Universal Robots PolyScope program: proiecFinalHILT_cri.urp

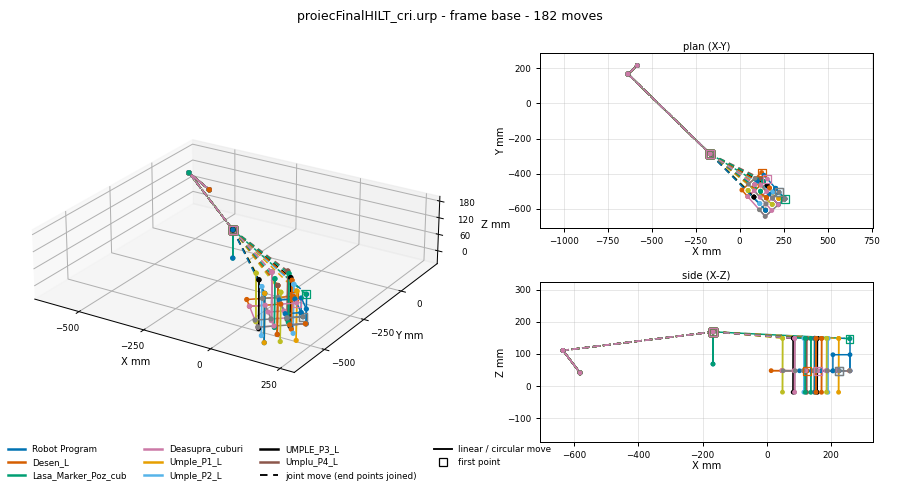
[picture p0: tool path of proiecFinalHILT_cri.urp in frame base, 182 of 182 moves have a stored position in this frame; points joined in program order, loops and branches not executed]
Program proiecFinalHILT_cri (installation=default directory=/home/ur/ursim-current/programs/Setup createdIn=3.15.5.106321 lastSavedIn=3.15.5.106321 robotSerialNumber=2018359999)
Calibrated DH parameters: a=[0, -0.425, -0.39225, 0, 0, 0]; d=[0.089159, 0, 0, 0.10915, 0.09465, 0.0823]; alpha=[1.570796, 0, 0, 1.570796, -1.570796, 0]; deltaTheta=[0, 0, 0, 0, 0, 0]
Robot Program (runOnlyOnce=false)
  MoveL speed 250 mm/s, acceleration 1200 mm/s^2 (useActiveTCP=true) feature=Base
    Waypoint Intermediar_cub: TCP in base x=-167.567 y=-286.499 z=168.811 mm, rx=1.2909 ry=2.8479 rz=-0.0144 rad; joints [39.36, -114.131, 107.649, -83.617, -89.01, -1.87] deg; flange x=-170.167 y=-282.588 z=439.18 mm, rx=1.2909 ry=2.8479 rz=-0.0144 rad
    Waypoint preluare_marker: TCP in base x=-167.81 y=-286.838 z=68.812 mm, rx=1.2909 ry=2.8479 rz=-0.0144 rad; joints [39.38, -113.83, 122.13, -98.4, -89.01, -1.85] deg; flange x=-170.409 y=-282.927 z=339.181 mm, rx=1.2909 ry=2.8479 rz=-0.0144 rad
    Wait Sleep waitTime=0.5
    'G 10'
    Wait Sleep waitTime=0.5
  MoveL speed 250 mm/s, acceleration 1200 mm/s^2 (useActiveTCP=true) feature=Base
    Waypoint ridicare_marker: TCP in base x=-167.568 y=-286.499 z=168.811 mm, rx=1.2909 ry=2.8479 rz=-0.0144 rad; joints [39.36, -114.131, 107.649, -83.617, -89.01, -1.87] deg; flange x=-170.167 y=-282.588 z=439.18 mm, rx=1.2909 ry=2.8479 rz=-0.0144 rad
  MoveJ speed 60 deg/s, acceleration 80 deg/s^2 (useActiveTCP=true)
    Waypoint deasupra_colt_f: TCP in base x=258.142 y=-542.024 z=147.75 mm, rx=1.296 ry=2.8485 rz=0.0145 rad; joints [104.471, -76.071, 76.258, -90.209, -89.13, 63.401] deg; flange x=254.141 y=-542.951 z=418.128 mm, rx=1.296 ry=2.8485 rz=0.0145 rad
  MoveL speed 250 mm/s, acceleration 1200 mm/s^2 (useActiveTCP=true) feature=Base
    Waypoint marker_pe_colt: TCP in base x=257.9 y=-542.363 z=47.75 mm, rx=1.296 ry=2.8485 rz=0.0145 rad; joints [104.44, -74.31, 88.769, -104.48, -89.13, 63.37] deg; flange x=253.899 y=-543.29 z=318.129 mm, rx=1.296 ry=2.8485 rz=0.0145 rad
  If digital_in[1] == True
    Call Desen_L
    Call Lasa_Marker_Poz_cub
    Call Deasupra_cuburi
    Call Umple_P1_L
    Call Umple_P2_L
    Call UMPLE_P3_L
    Call Umplu_P4_L
    Call Umplu_P5_L
    Call Umplu_P6_L
  If digital_in[2] ==  True
    Call Desen_i
    Call Lasa_Marker_Poz_cub
    Call Deasupra_cuburi
    Call Umple_P1_L
    Call Umplu_p2_i
    Call Umplu_p3_i
  If digital_in[3] ==  True
    Call Desen_H
    Call Lasa_Marker_Poz_cub
    Call Deasupra_cuburi
    Call Umple_P1_L
    Call Umple_P2_L
    Call UMPLE_P3_L
    Call Umple_P4_H
    Call Umple_P5_H
    Call Umple_P6_H
    Call Umple_P7_H
  If digital_in[5] ==  True
    Call Desen_T
    Call Lasa_Marker_Poz_cub
    Call Deasupra_cuburi
    Call Umple_P1_L
    Call Umple_P2_T
    Call Umple_p3_T
    Call Umplu_p4_t
    Call Umplu_p5_T
    Call Umple_P6_T
SubProgram -> Umple_P7_H
SubProgram -> Umple_P6_H
SubProgram -> Umple_P5_H
SubProgram -> Umple_P4_H
SubProgram -> Umple_P6_T
SubProgram -> Umplu_p5_T
SubProgram -> Umplu_p4_t
SubProgram -> Umple_p3_T
SubProgram -> Umple_P2_T
SubProgram -> Desen_H
SubProgram -> Desen_T
SubProgram -> Umplu_p3_i
SubProgram -> Umplu_p2_i
SubProgram -> Desen_i
SubProgram -> Umplu_P6_L
SubProgram -> Umplu_P5_L
SubProgram -> Umplu_P4_L
SubProgram -> UMPLE_P3_L
SubProgram -> Umple_P2_L
SubProgram -> Umple_P1_L
SubProgram -> Deasupra_cuburi
SubProgram -> Lasa_Marker_Poz_cub
SubProgram -> Desen_L
SubProgram Desen_L (keepSynchronizedWithDisk=false)
  MoveL speed 250 mm/s, acceleration 1200 mm/s^2 (useActiveTCP=true) feature=Base
    Waypoint exterior_L: TCP in base x=125.172 y=-392.753 z=47.565 mm, rx=1.296 ry=2.8485 rz=0.0145 rad; joints [91.565, -100.156, 115.983, -105.654, -89.147, 50.493] deg; flange x=121.171 y=-393.68 z=317.944 mm, rx=1.296 ry=2.8485 rz=0.0145 rad
  MoveL speed 250 mm/s, acceleration 1200 mm/s^2 (useActiveTCP=true) feature=Base
    Waypoint Exterior_L2: TCP in base x=12.964 y=-492.297 z=48.174 mm, rx=1.296 ry=2.8485 rz=0.0145 rad; joints [78.123, -88.524, 105.201, -106.311, -89.211, 37.05] deg; flange x=8.963 y=-493.224 z=318.552 mm, rx=1.296 ry=2.8485 rz=0.0145 rad
  MoveL speed 250 mm/s, acceleration 1200 mm/s^2 (useActiveTCP=true) feature=Base
    Waypoint Exterior_L3: TCP in base x=46.146 y=-529.7 z=48.22 mm, rx=1.296 ry=2.8485 rz=0.0145 rad; joints [82.58, -83.248, 99.507, -105.954, -89.185, 41.507] deg; flange x=42.145 y=-530.627 z=318.599 mm, rx=1.296 ry=2.8485 rz=0.0145 rad
  MoveL speed 250 mm/s, acceleration 1200 mm/s^2 (useActiveTCP=true) feature=Base
    Waypoint Interior_L: TCP in base x=120.04 y=-464.145 z=47.819 mm, rx=1.296 ry=2.8485 rz=0.0145 rad; joints [90.697, -90.465, 107.261, -106.61, -89.15, 49.626] deg; flange x=116.039 y=-465.073 z=318.198 mm, rx=1.296 ry=2.8485 rz=0.0145 rad
  MoveL speed 250 mm/s, acceleration 1200 mm/s^2 (useActiveTCP=true) feature=Base
    Waypoint Interior_L2: TCP in base x=219.586 y=-576.353 z=47.958 mm, rx=1.296 ry=2.8485 rz=0.0145 rad; joints [100.158, -72.107, 85.808, -103.657, -89.131, 59.087] deg; flange x=215.585 y=-577.28 z=318.337 mm, rx=1.296 ry=2.8485 rz=0.0145 rad
  MoveL speed 250 mm/s, acceleration 1200 mm/s^2 (useActiveTCP=true) feature=Base
    Waypoint Interior_L3: TCP in base x=256.233 y=-543.842 z=47.759 mm, rx=1.296 ry=2.8485 rz=0.0145 rad; joints [104.247, -74.225, 88.656, -104.449, -89.13, 63.177] deg; flange x=252.231 y=-544.769 z=318.138 mm, rx=1.296 ry=2.8485 rz=0.0145 rad
SubProgram Lasa_Marker_Poz_cub (keepSynchronizedWithDisk=false)
  MoveL speed 250 mm/s, acceleration 1200 mm/s^2 (useActiveTCP=true) feature=Base
    Waypoint DeasupraFoaie: TCP in base x=256.475 y=-543.503 z=147.759 mm, rx=1.296 ry=2.8485 rz=0.0145 rad; joints [104.278, -75.981, 76.142, -90.18, -89.13, 63.208] deg; flange x=252.473 y=-544.43 z=418.137 mm, rx=1.296 ry=2.8485 rz=0.0145 rad
  MoveJ speed 60 deg/s, acceleration 80 deg/s^2 (useActiveTCP=true)
    Waypoint DeasupraMarker: TCP in base x=-167.557 y=-286.49 z=168.795 mm, rx=1.2909 ry=2.8479 rz=-0.0143 rad; joints [39.36, -114.132, 107.651, -83.617, -89.01, -1.87] deg; flange x=-170.163 y=-282.585 z=439.164 mm, rx=1.2909 ry=2.8479 rz=-0.0143 rad
  MoveL speed 250 mm/s, acceleration 1200 mm/s^2 (useActiveTCP=true) feature=Base
    Waypoint LasaMarker: TCP in base x=-167.799 y=-286.829 z=68.796 mm, rx=1.2909 ry=2.8479 rz=-0.0143 rad; joints [39.38, -113.83, 122.132, -98.4, -89.01, -1.85] deg; flange x=-170.405 y=-282.924 z=339.165 mm, rx=1.2909 ry=2.8479 rz=-0.0143 rad
    Wait Sleep waitTime=0.5
    'G 40'
    Wait Sleep waitTime=0.5
  MoveL speed 250 mm/s, acceleration 1200 mm/s^2 (useActiveTCP=true) feature=Base
    Waypoint DeasupraMarker2: TCP in base x=-167.557 y=-286.49 z=168.795 mm, rx=1.2909 ry=2.8479 rz=-0.0143 rad; joints [39.36, -114.132, 107.651, -83.617, -89.01, -1.87] deg; flange x=-170.163 y=-282.585 z=439.164 mm, rx=1.2909 ry=2.8479 rz=-0.0143 rad
    Wait Sleep waitTime=0.5
    'G80'
SubProgram Deasupra_cuburi (keepSynchronizedWithDisk=false)
  MoveL speed 250 mm/s, acceleration 1200 mm/s^2 (useActiveTCP=true) feature=Base
    Waypoint DeasupraMarker2: TCP in base x=-167.557 y=-286.49 z=168.795 mm, rx=1.2909 ry=2.8479 rz=-0.0143 rad; joints [39.36, -114.132, 107.651, -83.617, -89.01, -1.87] deg; flange x=-170.163 y=-282.585 z=439.164 mm, rx=1.2909 ry=2.8479 rz=-0.0143 rad
  MoveJ speed 60 deg/s, acceleration 80 deg/s^2 (useActiveTCP=true)
    Waypoint poz_intermcub: TCP in base x=-634.049 y=166.753 z=111.017 mm, rx=1.0761 ry=2.3886 rz=1.0065 rad; joints [-7.715, -31.545, 17.047, -40.87, -122.454, -38.841] deg; flange x=-782.032 y=40.366 z=298.765 mm, rx=1.0761 ry=2.3886 rz=1.0065 rad
  MoveL speed 250 mm/s, acceleration 1200 mm/s^2 (useActiveTCP=true) feature=Base
    Waypoint prindere_cub: TCP in base x=-580.967 y=215.041 z=41.371 mm, rx=1.0761 ry=2.3886 rz=1.0065 rad; joints [-11.8, -45.21, 53.1, -65.52, -124.71, -42.93] deg; flange x=-728.95 y=88.654 z=229.118 mm, rx=1.0761 ry=2.3886 rz=1.0065 rad
    Wait Sleep waitTime=0.5
    'G40'
  MoveL speed 250 mm/s, acceleration 1200 mm/s^2 (useActiveTCP=true) feature=Base
    Waypoint poz_intermcub: TCP in base x=-634.049 y=166.753 z=111.017 mm, rx=1.0761 ry=2.3886 rz=1.0065 rad; joints [-7.715, -31.545, 17.047, -40.87, -122.454, -38.841] deg; flange x=-782.032 y=40.366 z=298.765 mm, rx=1.0761 ry=2.3886 rz=1.0065 rad
    Wait Sleep waitTime=0.5
SubProgram Umple_P1_L (keepSynchronizedWithDisk=false)
  MoveJ speed 60 deg/s, acceleration 80 deg/s^2 (useActiveTCP=true)
    Waypoint Intermediar_cub: TCP in base x=-167.567 y=-286.499 z=168.811 mm, rx=1.2909 ry=2.8479 rz=-0.0144 rad; joints [39.36, -114.131, 107.649, -83.617, -89.01, -1.87] deg; flange x=-170.167 y=-282.588 z=439.18 mm, rx=1.2909 ry=2.8479 rz=-0.0144 rad
    Wait Sleep waitTime=0.5
  MoveJ speed 60 deg/s, acceleration 80 deg/s^2 (useActiveTCP=true)
    Waypoint cb_deas_fo_cent: TCP in base x=222.984 y=-540.437 z=148.398 mm, rx=2.9837 ry=0.9733 rz=-0.0052 rad; joints [101.765, -78.264, 78.922, -90.858, -90.17, 155.632] deg; flange x=223.577 y=-539.348 z=418.805 mm, rx=2.9837 ry=0.9733 rz=-0.0052 rad
    Wait Sleep waitTime=0.5
  MoveL speed 250 mm/s, acceleration 1200 mm/s^2 (useActiveTCP=true) feature=Base
    Waypoint las_1_cub_foaie: TCP in base x=222.579 y=-541.004 z=-18.947 mm, rx=2.9837 ry=0.9733 rz=-0.0052 rad; joints [101.714, -73.294, 97.815, -114.721, -90.17, 155.581] deg; flange x=223.172 y=-539.915 z=251.46 mm, rx=2.9837 ry=0.9733 rz=-0.0052 rad
    Wait Sleep waitTime=0.5
    'G 80'
  MoveL speed 250 mm/s, acceleration 1200 mm/s^2 (useActiveTCP=true) feature=Base
    Waypoint Deasupra_foaiee: TCP in base x=222.984 y=-540.437 z=148.398 mm, rx=2.9837 ry=0.9733 rz=-0.0052 rad; joints [101.765, -78.264, 78.922, -90.858, -90.17, 155.632] deg; flange x=223.577 y=-539.348 z=418.805 mm, rx=2.9837 ry=0.9733 rz=-0.0052 rad
SubProgram Umple_P2_L (keepSynchronizedWithDisk=false)
  MoveJ speed 60 deg/s, acceleration 80 deg/s^2 (useActiveTCP=true)
    Waypoint interm_P2: TCP in base x=-167.567 y=-286.499 z=168.811 mm, rx=1.2909 ry=2.8479 rz=-0.0144 rad; joints [39.36, -114.131, 107.649, -83.617, -89.01, -1.87] deg; flange x=-170.167 y=-282.588 z=439.18 mm, rx=1.2909 ry=2.8479 rz=-0.0144 rad
    Wait Sleep waitTime=0.5
  MoveJ speed 60 deg/s, acceleration 80 deg/s^2 (useActiveTCP=true)
    Waypoint DEAS_cub_C2_L: TCP in base x=-634.049 y=166.753 z=111.017 mm, rx=1.0761 ry=2.3886 rz=1.0065 rad; joints [-7.715, -31.545, 17.047, -40.87, -122.454, -38.841] deg; flange x=-782.032 y=40.366 z=298.765 mm, rx=1.0761 ry=2.3886 rz=1.0065 rad
    Wait Sleep waitTime=0.5
  MoveL speed 250 mm/s, acceleration 1200 mm/s^2 (useActiveTCP=true) feature=Base
    Waypoint prel_c2_L: TCP in base x=-580.967 y=215.041 z=41.371 mm, rx=1.0761 ry=2.3886 rz=1.0065 rad; joints [-11.8, -45.21, 53.1, -65.52, -124.71, -42.93] deg; flange x=-728.95 y=88.654 z=229.118 mm, rx=1.0761 ry=2.3886 rz=1.0065 rad
    Wait Sleep waitTime=0.5
    'G40'
  MoveL speed 250 mm/s, acceleration 1200 mm/s^2 (useActiveTCP=true) feature=Base
    Waypoint deas_c2_L: TCP in base x=-634.049 y=166.753 z=111.017 mm, rx=1.0761 ry=2.3886 rz=1.0065 rad; joints [-7.715, -31.545, 17.047, -40.87, -122.454, -38.841] deg; flange x=-782.032 y=40.366 z=298.765 mm, rx=1.0761 ry=2.3886 rz=1.0065 rad
    Wait Sleep waitTime=0.5
  MoveJ speed 60 deg/s, acceleration 80 deg/s^2 (useActiveTCP=true)
    Waypoint INTERM: TCP in base x=-167.567 y=-286.499 z=168.811 mm, rx=1.2909 ry=2.8479 rz=-0.0144 rad; joints [39.36, -114.131, 107.649, -83.617, -89.01, -1.87] deg; flange x=-170.167 y=-282.588 z=439.18 mm, rx=1.2909 ry=2.8479 rz=-0.0144 rad
    Wait Sleep waitTime=0.5
  MoveJ speed 60 deg/s, acceleration 80 deg/s^2 (useActiveTCP=true)
    Waypoint DEAS_P2_L_FOAIE: TCP in base x=189.802 y=-503.035 z=148.352 mm, rx=2.9837 ry=0.9733 rz=-0.0052 rad; joints [99.066, -84.782, 86.489, -91.915, -90.16, 152.933] deg; flange x=190.395 y=-501.946 z=418.759 mm, rx=2.9837 ry=0.9733 rz=-0.0052 rad
    Wait Sleep waitTime=0.5
  MoveL speed 250 mm/s, acceleration 1200 mm/s^2 (useActiveTCP=true) feature=Base
    Waypoint LAS_P2_L_FOAIE: TCP in base x=189.397 y=-503.602 z=-18.994 mm, rx=2.9837 ry=0.9733 rz=-0.0052 rad; joints [99.013, -79.253, 105.478, -116.434, -90.16, 152.88] deg; flange x=189.99 y=-502.512 z=251.414 mm, rx=2.9837 ry=0.9733 rz=-0.0052 rad
    Wait Sleep waitTime=0.5
    'G 80'
  MoveL speed 250 mm/s, acceleration 1200 mm/s^2 (useActiveTCP=true) feature=Base
    Waypoint DEAS_P2_L: TCP in base x=189.802 y=-503.035 z=148.352 mm, rx=2.9837 ry=0.9733 rz=-0.0052 rad; joints [99.067, -84.782, 86.489, -91.915, -90.16, 152.933] deg; flange x=190.395 y=-501.945 z=418.759 mm, rx=2.9837 ry=0.9733 rz=-0.0052 rad
SubProgram UMPLE_P3_L (keepSynchronizedWithDisk=false)
  MoveJ speed 60 deg/s, acceleration 80 deg/s^2 (useActiveTCP=true)
    Waypoint INTERM_P3: TCP in base x=-167.567 y=-286.499 z=168.811 mm, rx=1.2909 ry=2.8479 rz=-0.0144 rad; joints [39.36, -114.131, 107.649, -83.617, -89.01, -1.87] deg; flange x=-170.167 y=-282.588 z=439.18 mm, rx=1.2909 ry=2.8479 rz=-0.0144 rad
    Wait Sleep waitTime=0.5
  MoveJ speed 60 deg/s, acceleration 80 deg/s^2 (useActiveTCP=true)
    Waypoint DEAS_C3_L: TCP in base x=-634.049 y=166.753 z=111.017 mm, rx=1.0761 ry=2.3886 rz=1.0065 rad; joints [-7.715, -31.545, 17.047, -40.87, -122.454, -38.841] deg; flange x=-782.032 y=40.366 z=298.765 mm, rx=1.0761 ry=2.3886 rz=1.0065 rad
    Wait Sleep waitTime=0.5
  MoveL speed 250 mm/s, acceleration 1200 mm/s^2 (useActiveTCP=true) feature=Base
    Waypoint PREL_C3_L: TCP in base x=-580.967 y=215.041 z=41.371 mm, rx=1.0761 ry=2.3886 rz=1.0065 rad; joints [-11.8, -45.21, 53.1, -65.52, -124.71, -42.93] deg; flange x=-728.95 y=88.654 z=229.118 mm, rx=1.0761 ry=2.3886 rz=1.0065 rad
    Wait Sleep waitTime=0.5
    'G40'
  MoveL speed 250 mm/s, acceleration 1200 mm/s^2 (useActiveTCP=true) feature=Base
    Waypoint DEAS_C3_LL: TCP in base x=-634.049 y=166.753 z=111.017 mm, rx=1.0761 ry=2.3886 rz=1.0065 rad; joints [-7.715, -31.545, 17.047, -40.87, -122.454, -38.841] deg; flange x=-782.032 y=40.366 z=298.765 mm, rx=1.0761 ry=2.3886 rz=1.0065 rad
    Wait Sleep waitTime=0.5
  MoveJ speed 60 deg/s, acceleration 80 deg/s^2 (useActiveTCP=true)
    Waypoint INTERMMM: TCP in base x=-167.567 y=-286.499 z=168.811 mm, rx=1.2909 ry=2.8479 rz=-0.0144 rad; joints [39.36, -114.131, 107.649, -83.617, -89.01, -1.87] deg; flange x=-170.167 y=-282.588 z=439.18 mm, rx=1.2909 ry=2.8479 rz=-0.0144 rad
    Wait Sleep waitTime=0.5
  MoveJ speed 60 deg/s, acceleration 80 deg/s^2 (useActiveTCP=true)
    Waypoint DEAS_P3_L_FOAIE: TCP in base x=156.62 y=-465.632 z=148.305 mm, rx=2.9837 ry=0.9733 rz=-0.0052 rad; joints [95.863, -91.188, 93.147, -92.177, -90.149, 149.73] deg; flange x=157.213 y=-464.543 z=418.713 mm, rx=2.9837 ry=0.9733 rz=-0.0052 rad
    Wait Sleep waitTime=0.5
  MoveL speed 250 mm/s, acceleration 1200 mm/s^2 (useActiveTCP=true) feature=Base
    Waypoint LAS_P3_L_FOAIE: TCP in base x=156.215 y=-466.199 z=-19.04 mm, rx=2.9837 ry=0.9733 rz=-0.0052 rad; joints [95.808, -85.301, 112.521, -117.438, -90.148, 149.675] deg; flange x=156.808 y=-465.11 z=251.367 mm, rx=2.9837 ry=0.9733 rz=-0.0052 rad
    Wait Sleep waitTime=0.5
    'G 80'
  MoveL speed 250 mm/s, acceleration 1200 mm/s^2 (useActiveTCP=true) feature=Base
    Waypoint DEASUPRA_P3_L: TCP in base x=156.62 y=-465.632 z=148.305 mm, rx=2.9837 ry=0.9733 rz=-0.0052 rad; joints [95.863, -91.188, 93.147, -92.177, -90.149, 149.73] deg; flange x=157.213 y=-464.543 z=418.713 mm, rx=2.9837 ry=0.9733 rz=-0.0052 rad
SubProgram Umplu_P4_L (keepSynchronizedWithDisk=false)
  MoveJ speed 60 deg/s, acceleration 80 deg/s^2 (useActiveTCP=true)
    Waypoint INTERM_P4: TCP in base x=-167.567 y=-286.499 z=168.811 mm, rx=1.2909 ry=2.8479 rz=-0.0144 rad; joints [39.36, -114.131, 107.649, -83.617, -89.01, -1.87] deg; flange x=-170.167 y=-282.588 z=439.18 mm, rx=1.2909 ry=2.8479 rz=-0.0144 rad
    Wait Sleep waitTime=0.5
  MoveJ speed 60 deg/s, acceleration 80 deg/s^2 (useActiveTCP=true)
    Waypoint DEAS_C4_L: TCP in base x=-634.049 y=166.753 z=111.017 mm, rx=1.0761 ry=2.3886 rz=1.0065 rad; joints [-7.715, -31.545, 17.047, -40.87, -122.454, -38.841] deg; flange x=-782.032 y=40.366 z=298.765 mm, rx=1.0761 ry=2.3886 rz=1.0065 rad
    Wait Sleep waitTime=0.5
  MoveL speed 250 mm/s, acceleration 1200 mm/s^2 (useActiveTCP=true) feature=Base
    Waypoint PREL_C4_L: TCP in base x=-580.967 y=215.041 z=41.371 mm, rx=1.0761 ry=2.3886 rz=1.0065 rad; joints [-11.8, -45.21, 53.1, -65.52, -124.71, -42.93] deg; flange x=-728.95 y=88.654 z=229.118 mm, rx=1.0761 ry=2.3886 rz=1.0065 rad
    Wait Sleep waitTime=0.5
    'G40'
  MoveL speed 250 mm/s, acceleration 1200 mm/s^2 (useActiveTCP=true) feature=Base
    Waypoint DEAS_C4_LL: TCP in base x=-634.049 y=166.753 z=111.017 mm, rx=1.0761 ry=2.3886 rz=1.0065 rad; joints [-7.715, -31.545, 17.047, -40.87, -122.454, -38.841] deg; flange x=-782.032 y=40.366 z=298.765 mm, rx=1.0761 ry=2.3886 rz=1.0065 rad
    Wait Sleep waitTime=0.5
  MoveJ speed 60 deg/s, acceleration 80 deg/s^2 (useActiveTCP=true)
    Waypoint INTER: TCP in base x=-167.567 y=-286.499 z=168.811 mm, rx=1.2909 ry=2.8479 rz=-0.0144 rad; joints [39.36, -114.131, 107.649, -83.617, -89.01, -1.87] deg; flange x=-170.167 y=-282.588 z=439.18 mm, rx=1.2909 ry=2.8479 rz=-0.0144 rad
    Wait Sleep waitTime=0.5
  MoveJ speed 60 deg/s, acceleration 80 deg/s^2 (useActiveTCP=true)
    Waypoint DEAS_P4_L_FOAIE: TCP in base x=123.438 y=-428.23 z=148.259 mm, rx=2.9837 ry=0.9733 rz=-0.0052 rad; joints [92.012, -97.554, 98.997, -91.67, -90.134, 145.879] deg; flange x=124.031 y=-427.14 z=418.666 mm, rx=2.9837 ry=0.9733 rz=-0.0052 rad
    Wait Sleep waitTime=0.5
  MoveL speed 250 mm/s, acceleration 1200 mm/s^2 (useActiveTCP=true) feature=Base
    Waypoint LAS_P4_L_FOAIE: TCP in base x=123.033 y=-428.796 z=-19.086 mm, rx=2.9837 ry=0.9733 rz=-0.0052 rad; joints [91.956, -91.539, 118.98, -117.667, -90.133, 145.823] deg; flange x=123.626 y=-427.707 z=251.321 mm, rx=2.9837 ry=0.9733 rz=-0.0052 rad
    Wait Sleep waitTime=0.5
    'G 80'
  MoveL speed 250 mm/s, acceleration 1200 mm/s^2 (useActiveTCP=true) feature=Base
    Waypoint DEAS_P4_L: TCP in base x=123.438 y=-428.23 z=148.259 mm, rx=2.9837 ry=0.9733 rz=-0.0052 rad; joints [92.012, -97.554, 98.997, -91.67, -90.134, 145.879] deg; flange x=124.031 y=-427.14 z=418.666 mm, rx=2.9837 ry=0.9733 rz=-0.0052 rad
SubProgram Umplu_P5_L (keepSynchronizedWithDisk=false)
  MoveJ speed 60 deg/s, acceleration 80 deg/s^2 (useActiveTCP=true)
    Waypoint INTERM_P5: TCP in base x=-167.567 y=-286.499 z=168.811 mm, rx=1.2909 ry=2.8479 rz=-0.0144 rad; joints [39.36, -114.131, 107.649, -83.617, -89.01, -1.87] deg; flange x=-170.167 y=-282.588 z=439.18 mm, rx=1.2909 ry=2.8479 rz=-0.0144 rad
    Wait Sleep waitTime=0.5
  MoveJ speed 60 deg/s, acceleration 80 deg/s^2 (useActiveTCP=true)
    Waypoint DEAS_C5_L: TCP in base x=-634.049 y=166.753 z=111.017 mm, rx=1.0761 ry=2.3886 rz=1.0065 rad; joints [-7.715, -31.545, 17.047, -40.87, -122.454, -38.841] deg; flange x=-782.032 y=40.366 z=298.765 mm, rx=1.0761 ry=2.3886 rz=1.0065 rad
    Wait Sleep waitTime=0.5
  MoveL speed 250 mm/s, acceleration 1200 mm/s^2 (useActiveTCP=true) feature=Base
    Waypoint PREL_C5_L: TCP in base x=-580.967 y=215.041 z=41.371 mm, rx=1.0761 ry=2.3886 rz=1.0065 rad; joints [-11.8, -45.21, 53.1, -65.52, -124.71, -42.93] deg; flange x=-728.95 y=88.654 z=229.118 mm, rx=1.0761 ry=2.3886 rz=1.0065 rad
    Wait Sleep waitTime=0.5
    'G40'
  MoveL speed 250 mm/s, acceleration 1200 mm/s^2 (useActiveTCP=true) feature=Base
    Waypoint DEAS_C5_LL: TCP in base x=-634.049 y=166.753 z=111.017 mm, rx=1.0761 ry=2.3886 rz=1.0065 rad; joints [-7.715, -31.545, 17.047, -40.87, -122.454, -38.841] deg; flange x=-782.032 y=40.366 z=298.765 mm, rx=1.0761 ry=2.3886 rz=1.0065 rad
    Wait Sleep waitTime=0.5
  MoveJ speed 60 deg/s, acceleration 80 deg/s^2 (useActiveTCP=true)
    Waypoint INTERR: TCP in base x=-167.567 y=-286.499 z=168.811 mm, rx=1.2909 ry=2.8479 rz=-0.0144 rad; joints [39.36, -114.131, 107.649, -83.617, -89.01, -1.87] deg; flange x=-170.167 y=-282.588 z=439.18 mm, rx=1.2909 ry=2.8479 rz=-0.0144 rad
    Wait Sleep waitTime=0.5
  MoveJ speed 60 deg/s, acceleration 80 deg/s^2 (useActiveTCP=true)
    Waypoint DEAS_P5_L_FOAIE: TCP in base x=86.036 y=-461.411 z=148.462 mm, rx=1.2912 ry=2.8474 rz=-0.0143 rad; joints [86.636, -94.863, 96.738, -92.673, -89.38, 45.427] deg; flange x=83.337 y=-457.477 z=418.83 mm, rx=1.2912 ry=2.8474 rz=-0.0143 rad
    Wait Sleep waitTime=0.5
  MoveL speed 250 mm/s, acceleration 1200 mm/s^2 (useActiveTCP=true) feature=Base
    Waypoint LAS_P5_L_FOAIE: TCP in base x=85.631 y=-461.978 z=-18.883 mm, rx=1.2912 ry=2.8474 rz=-0.0143 rad; joints [86.589, -88.809, 116.39, -118.379, -89.38, 45.38] deg; flange x=82.932 y=-458.043 z=251.485 mm, rx=1.2912 ry=2.8474 rz=-0.0143 rad
    Wait Sleep waitTime=0.5
    'G 80'
  MoveL speed 250 mm/s, acceleration 1200 mm/s^2 (useActiveTCP=true) feature=Base
    Waypoint DEAS_P5_L: TCP in base x=86.036 y=-461.411 z=148.462 mm, rx=1.2912 ry=2.8474 rz=-0.0143 rad; joints [86.636, -94.863, 96.738, -92.673, -89.38, 45.427] deg; flange x=83.337 y=-457.477 z=418.83 mm, rx=1.2912 ry=2.8474 rz=-0.0143 rad
SubProgram Umplu_P6_L (keepSynchronizedWithDisk=false)
  MoveJ speed 60 deg/s, acceleration 80 deg/s^2 (useActiveTCP=true)
    Waypoint INTERM_P6: TCP in base x=-167.567 y=-286.499 z=168.811 mm, rx=1.2909 ry=2.8479 rz=-0.0144 rad; joints [39.36, -114.131, 107.649, -83.617, -89.01, -1.87] deg; flange x=-170.167 y=-282.588 z=439.18 mm, rx=1.2909 ry=2.8479 rz=-0.0144 rad
    Wait Sleep waitTime=0.5
  MoveJ speed 60 deg/s, acceleration 80 deg/s^2 (useActiveTCP=true)
    Waypoint DEAS_C6_L: TCP in base x=-634.049 y=166.753 z=111.017 mm, rx=1.0761 ry=2.3886 rz=1.0065 rad; joints [-7.715, -31.545, 17.047, -40.87, -122.454, -38.841] deg; flange x=-782.032 y=40.366 z=298.765 mm, rx=1.0761 ry=2.3886 rz=1.0065 rad
    Wait Sleep waitTime=0.5
  MoveL speed 250 mm/s, acceleration 1200 mm/s^2 (useActiveTCP=true) feature=Base
    Waypoint PREL_C6_L: TCP in base x=-580.967 y=215.041 z=41.371 mm, rx=1.0761 ry=2.3886 rz=1.0065 rad; joints [-11.8, -45.21, 53.1, -65.52, -124.71, -42.93] deg; flange x=-728.95 y=88.654 z=229.118 mm, rx=1.0761 ry=2.3886 rz=1.0065 rad
    Wait Sleep waitTime=0.5
    'G40'
  MoveL speed 250 mm/s, acceleration 1200 mm/s^2 (useActiveTCP=true) feature=Base
    Waypoint DEAS_C6_LL: TCP in base x=-634.049 y=166.753 z=111.017 mm, rx=1.0761 ry=2.3886 rz=1.0065 rad; joints [-7.715, -31.545, 17.047, -40.87, -122.454, -38.841] deg; flange x=-782.032 y=40.366 z=298.765 mm, rx=1.0761 ry=2.3886 rz=1.0065 rad
    Wait Sleep waitTime=0.5
  MoveJ speed 60 deg/s, acceleration 80 deg/s^2 (useActiveTCP=true)
    Waypoint INTERRR: TCP in base x=-167.567 y=-286.499 z=168.811 mm, rx=1.2909 ry=2.8479 rz=-0.0144 rad; joints [39.36, -114.131, 107.649, -83.617, -89.01, -1.87] deg; flange x=-170.167 y=-282.588 z=439.18 mm, rx=1.2909 ry=2.8479 rz=-0.0144 rad
    Wait Sleep waitTime=0.5
  MoveJ speed 60 deg/s, acceleration 80 deg/s^2 (useActiveTCP=true)
    Waypoint DEAS_P6_L_FOAIE: TCP in base x=48.634 y=-494.593 z=148.665 mm, rx=1.2912 ry=2.8474 rz=-0.0143 rad; joints [82.436, -90.995, 93.042, -92.799, -89.323, 41.227] deg; flange x=45.935 y=-490.658 z=419.033 mm, rx=1.2912 ry=2.8474 rz=-0.0143 rad
    Wait Sleep waitTime=0.5
  MoveL speed 250 mm/s, acceleration 1200 mm/s^2 (useActiveTCP=true) feature=Base
    Waypoint LAS_C6_L_FOAIE: TCP in base x=48.228 y=-495.159 z=-18.68 mm, rx=1.2912 ry=2.8474 rz=-0.0143 rad; joints [82.397, -85.063, 112.354, -118.041, -89.323, 41.188] deg; flange x=45.53 y=-491.225 z=251.687 mm, rx=1.2912 ry=2.8474 rz=-0.0143 rad
    Wait Sleep waitTime=0.5
    'G 80'
  MoveL speed 250 mm/s, acceleration 1200 mm/s^2 (useActiveTCP=true) feature=Base
    Waypoint DEAS_P6_L: TCP in base x=48.634 y=-494.593 z=148.665 mm, rx=1.2912 ry=2.8474 rz=-0.0143 rad; joints [82.436, -90.995, 93.042, -92.799, -89.323, 41.227] deg; flange x=45.935 y=-490.659 z=419.033 mm, rx=1.2912 ry=2.8474 rz=-0.0143 rad
SubProgram Desen_i (keepSynchronizedWithDisk=false)
  MoveL speed 250 mm/s, acceleration 1200 mm/s^2 (useActiveTCP=true) feature=Base
    Waypoint Caciulita_i1: TCP in base x=224.718 y=-504.96 z=47.704 mm, rx=1.2912 ry=2.8474 rz=-0.0143 rad; joints [102.353, -81.264, 97.613, -107.286, -89.62, 61.142] deg; flange x=222.019 y=-501.026 z=318.072 mm, rx=1.2912 ry=2.8474 rz=-0.0143 rad
  MoveL speed 250 mm/s, acceleration 1200 mm/s^2 (useActiveTCP=true) feature=Base
    Waypoint Caciulita_i2: TCP in base x=187.315 y=-538.142 z=47.907 mm, rx=1.2912 ry=2.8474 rz=-0.0143 rad; joints [97.863, -78.985, 94.854, -106.774, -89.548, 56.653] deg; flange x=184.617 y=-534.208 z=318.275 mm, rx=1.2912 ry=2.8474 rz=-0.0143 rad
  MoveL speed 250 mm/s, acceleration 1200 mm/s^2 (useActiveTCP=true) feature=Base
    Waypoint caciulita_i3: TCP in base x=220.497 y=-575.545 z=47.954 mm, rx=1.2912 ry=2.8474 rz=-0.0143 rad; joints [100.523, -72.822, 87.007, -105.109, -89.59, 59.313] deg; flange x=217.799 y=-571.61 z=318.321 mm, rx=1.2912 ry=2.8474 rz=-0.0143 rad
  MoveL speed 250 mm/s, acceleration 1200 mm/s^2 (useActiveTCP=true) feature=Base
    Waypoint Caciulita_i4: TCP in base x=257.9 y=-542.363 z=47.75 mm, rx=1.2912 ry=2.8474 rz=-0.0143 rad; joints [104.757, -74.921, 89.796, -105.827, -89.659, 63.546] deg; flange x=255.201 y=-538.429 z=318.118 mm, rx=1.2912 ry=2.8474 rz=-0.0143 rad
  MoveL speed 250 mm/s, acceleration 1200 mm/s^2 (useActiveTCP=true) feature=Base
    Waypoint spatiere1_i: TCP in base x=258.021 y=-542.194 z=97.75 mm, rx=1.2912 ry=2.8474 rz=-0.0143 rad; joints [104.772, -76.261, 84.051, -98.742, -89.66, 63.562] deg; flange x=255.322 y=-538.259 z=368.118 mm, rx=1.2912 ry=2.8474 rz=-0.0143 rad
  MoveL speed 250 mm/s, acceleration 1200 mm/s^2 (useActiveTCP=true) feature=Base
    Waypoint spatiere2_i: TCP in base x=204.93 y=-482.35 z=97.676 mm, rx=1.2912 ry=2.8474 rz=-0.0143 rad; joints [100.717, -86.652, 96.136, -100.409, -89.593, 59.508] deg; flange x=202.231 y=-478.415 z=368.044 mm, rx=1.2912 ry=2.8474 rz=-0.0143 rad
  MoveL speed 250 mm/s, acceleration 1200 mm/s^2 (useActiveTCP=true) feature=Base
    Waypoint spatiere3_i: TCP in base x=204.809 y=-482.519 z=47.676 mm, rx=1.2912 ry=2.8474 rz=-0.0143 rad; joints [100.7, -85.081, 101.945, -107.789, -89.593, 59.491] deg; flange x=202.11 y=-478.584 z=318.044 mm, rx=1.2912 ry=2.8474 rz=-0.0143 rad
  MoveL speed 250 mm/s, acceleration 1200 mm/s^2 (useActiveTCP=true) feature=Base
    Waypoint coada_i1: TCP in base x=138.445 y=-407.714 z=47.584 mm, rx=1.2912 ry=2.8474 rz=-0.0143 rad; joints [93.632, -98.188, 114.63, -107.31, -89.482, 52.423] deg; flange x=135.746 y=-403.779 z=317.952 mm, rx=1.2912 ry=2.8474 rz=-0.0143 rad
  MoveL speed 250 mm/s, acceleration 1200 mm/s^2 (useActiveTCP=true) feature=Base
    Waypoint coada_i2: TCP in base x=101.042 y=-440.895 z=47.787 mm, rx=1.2912 ry=2.8474 rz=-0.0143 rad; joints [88.466, -95.012, 111.823, -107.629, -89.406, 47.257] deg; flange x=98.344 y=-436.961 z=318.155 mm, rx=1.2912 ry=2.8474 rz=-0.0143 rad
  MoveL speed 250 mm/s, acceleration 1200 mm/s^2 (useActiveTCP=true) feature=Base
    Waypoint coada_i3: TCP in base x=167.406 y=-515.7 z=47.879 mm, rx=1.2912 ry=2.8474 rz=-0.0143 rad; joints [96.051, -82.656, 99.187, -107.42, -89.519, 54.842] deg; flange x=164.708 y=-511.766 z=318.247 mm, rx=1.2912 ry=2.8474 rz=-0.0143 rad
  MoveL speed 250 mm/s, acceleration 1200 mm/s^2 (useActiveTCP=true) feature=Base
    Waypoint coada_i4: TCP in base x=204.809 y=-482.519 z=47.677 mm, rx=1.2912 ry=2.8474 rz=-0.0143 rad; joints [100.7, -85.081, 101.945, -107.789, -89.593, 59.491] deg; flange x=202.11 y=-478.584 z=318.045 mm, rx=1.2912 ry=2.8474 rz=-0.0143 rad
SubProgram Umplu_p2_i (keepSynchronizedWithDisk=false)
  MoveJ speed 60 deg/s, acceleration 80 deg/s^2 (useActiveTCP=true)
    Waypoint interm_p2_i: TCP in base x=-167.567 y=-286.499 z=168.811 mm, rx=1.2909 ry=2.8479 rz=-0.0144 rad; joints [39.36, -114.131, 107.649, -83.617, -89.01, -1.87] deg; flange x=-170.167 y=-282.588 z=439.18 mm, rx=1.2909 ry=2.8479 rz=-0.0144 rad
    Wait Sleep waitTime=0.5
  MoveJ speed 60 deg/s, acceleration 80 deg/s^2 (useActiveTCP=true)
    Waypoint deas_c2_i: TCP in base x=-634.049 y=166.753 z=111.017 mm, rx=1.0761 ry=2.3886 rz=1.0065 rad; joints [-7.715, -31.545, 17.047, -40.87, -122.454, -38.841] deg; flange x=-782.032 y=40.366 z=298.765 mm, rx=1.0761 ry=2.3886 rz=1.0065 rad
    Wait Sleep waitTime=0.5
  MoveL speed 250 mm/s, acceleration 1200 mm/s^2 (useActiveTCP=true) feature=Base
    Waypoint prel_c2_i: TCP in base x=-580.967 y=215.041 z=41.371 mm, rx=1.0761 ry=2.3886 rz=1.0065 rad; joints [-11.8, -45.21, 53.1, -65.52, -124.71, -42.93] deg; flange x=-728.95 y=88.654 z=229.118 mm, rx=1.0761 ry=2.3886 rz=1.0065 rad
    Wait Sleep waitTime=0.5
    'G40'
  MoveL speed 250 mm/s, acceleration 1200 mm/s^2 (useActiveTCP=true) feature=Base
    Waypoint deas_c2_i2: TCP in base x=-634.049 y=166.753 z=111.017 mm, rx=1.0761 ry=2.3886 rz=1.0065 rad; joints [-7.715, -31.545, 17.047, -40.87, -122.454, -38.841] deg; flange x=-782.032 y=40.366 z=298.765 mm, rx=1.0761 ry=2.3886 rz=1.0065 rad
    Wait Sleep waitTime=0.5
  MoveJ speed 60 deg/s, acceleration 80 deg/s^2 (useActiveTCP=true)
    Waypoint intermmm: TCP in base x=-167.567 y=-286.499 z=168.811 mm, rx=1.2909 ry=2.8479 rz=-0.0144 rad; joints [39.36, -114.131, 107.649, -83.617, -89.01, -1.87] deg; flange x=-170.167 y=-282.588 z=439.18 mm, rx=1.2909 ry=2.8479 rz=-0.0144 rad
    Wait Sleep waitTime=0.5
  MoveJ speed 60 deg/s, acceleration 80 deg/s^2 (useActiveTCP=true)
    Waypoint Deas_P2_I_FOaie: TCP in base x=169.893 y=-480.593 z=148.324 mm, rx=2.9837 ry=0.9733 rz=-0.0052 rad; joints [97.213, -88.633, 90.585, -92.165, -90.154, 151.08] deg; flange x=170.486 y=-479.504 z=418.731 mm, rx=2.9837 ry=0.9733 rz=-0.0052 rad
    Wait Sleep waitTime=0.5
  MoveL speed 250 mm/s, acceleration 1200 mm/s^2 (useActiveTCP=true) feature=Base
    Waypoint las_P2_i_foaie: TCP in base x=169.488 y=-481.16 z=-19.021 mm, rx=2.9837 ry=0.9733 rz=-0.0052 rad; joints [97.159, -82.864, 109.775, -117.124, -90.153, 151.026] deg; flange x=170.081 y=-480.071 z=251.386 mm, rx=2.9837 ry=0.9733 rz=-0.0052 rad
    Wait Sleep waitTime=0.5
    'G 80'
  MoveL speed 250 mm/s, acceleration 1200 mm/s^2 (useActiveTCP=true) feature=Base
    Waypoint deas_p2_i: TCP in base x=169.893 y=-480.593 z=148.324 mm, rx=2.9837 ry=0.9733 rz=-0.0052 rad; joints [97.213, -88.633, 90.585, -92.165, -90.154, 151.08] deg; flange x=170.486 y=-479.504 z=418.731 mm, rx=2.9837 ry=0.9733 rz=-0.0052 rad
SubProgram Umplu_p3_i (keepSynchronizedWithDisk=false)
  MoveJ speed 60 deg/s, acceleration 80 deg/s^2 (useActiveTCP=true)
    Waypoint interm_p3: TCP in base x=-167.567 y=-286.499 z=168.811 mm, rx=1.2909 ry=2.8479 rz=-0.0144 rad; joints [39.36, -114.131, 107.649, -83.617, -89.01, -1.87] deg; flange x=-170.167 y=-282.588 z=439.18 mm, rx=1.2909 ry=2.8479 rz=-0.0144 rad
    Wait Sleep waitTime=0.5
  MoveJ speed 60 deg/s, acceleration 80 deg/s^2 (useActiveTCP=true)
    Waypoint deas_c3_i: TCP in base x=-634.049 y=166.753 z=111.017 mm, rx=1.0761 ry=2.3886 rz=1.0065 rad; joints [-7.715, -31.545, 17.047, -40.87, -122.454, -38.841] deg; flange x=-782.032 y=40.366 z=298.765 mm, rx=1.0761 ry=2.3886 rz=1.0065 rad
    Wait Sleep waitTime=0.5
  MoveL speed 250 mm/s, acceleration 1200 mm/s^2 (useActiveTCP=true) feature=Base
    Waypoint prel_3_i: TCP in base x=-580.967 y=215.041 z=41.371 mm, rx=1.0761 ry=2.3886 rz=1.0065 rad; joints [-11.8, -45.21, 53.1, -65.52, -124.71, -42.93] deg; flange x=-728.95 y=88.654 z=229.118 mm, rx=1.0761 ry=2.3886 rz=1.0065 rad
    Wait Sleep waitTime=0.5
    'G40'
  MoveL speed 250 mm/s, acceleration 1200 mm/s^2 (useActiveTCP=true) feature=Base
    Waypoint deas_c3_ii: TCP in base x=-634.049 y=166.753 z=111.017 mm, rx=1.0761 ry=2.3886 rz=1.0065 rad; joints [-7.715, -31.545, 17.047, -40.87, -122.454, -38.841] deg; flange x=-782.032 y=40.366 z=298.765 mm, rx=1.0761 ry=2.3886 rz=1.0065 rad
    Wait Sleep waitTime=0.5
  MoveJ speed 60 deg/s, acceleration 80 deg/s^2 (useActiveTCP=true)
    Waypoint interm: TCP in base x=-167.567 y=-286.499 z=168.811 mm, rx=1.2909 ry=2.8479 rz=-0.0144 rad; joints [39.36, -114.131, 107.649, -83.617, -89.01, -1.87] deg; flange x=-170.167 y=-282.588 z=439.18 mm, rx=1.2909 ry=2.8479 rz=-0.0144 rad
    Wait Sleep waitTime=0.5
  MoveJ speed 60 deg/s, acceleration 80 deg/s^2 (useActiveTCP=true)
    Waypoint deas_p3_i_foaie: TCP in base x=136.711 y=-443.191 z=148.278 mm, rx=2.9837 ry=0.9733 rz=-0.0052 rad; joints [93.641, -95.009, 96.75, -91.964, -90.14, 147.508] deg; flange x=137.304 y=-442.101 z=418.685 mm, rx=2.9837 ry=0.9733 rz=-0.0052 rad
    Wait Sleep waitTime=0.5
  MoveL speed 250 mm/s, acceleration 1200 mm/s^2 (useActiveTCP=true) feature=Base
    Waypoint las_p3_i_foaie: TCP in base x=136.306 y=-443.757 z=-19.068 mm, rx=2.9837 ry=0.9733 rz=-0.0052 rad; joints [93.585, -89.014, 116.466, -117.674, -90.14, 147.452] deg; flange x=136.899 y=-442.668 z=251.339 mm, rx=2.9837 ry=0.9733 rz=-0.0052 rad
    Wait Sleep waitTime=0.5
    'G 80'
  MoveL speed 250 mm/s, acceleration 1200 mm/s^2 (useActiveTCP=true) feature=Base
    Waypoint deas_p3_i: TCP in base x=136.711 y=-443.191 z=148.278 mm, rx=2.9837 ry=0.9733 rz=-0.0052 rad; joints [93.641, -95.009, 96.75, -91.964, -90.14, 147.508] deg; flange x=137.304 y=-442.101 z=418.685 mm, rx=2.9837 ry=0.9733 rz=-0.0052 rad
SubProgram Desen_H (keepSynchronizedWithDisk=false)
  MoveL speed 250 mm/s, acceleration 1200 mm/s^2 (useActiveTCP=true) feature=Base
    Waypoint L1_H: TCP in base x=158.354 y=-430.155 z=47.611 mm, rx=1.296 ry=2.8485 rz=0.0145 rad; joints [95.75, -93.475, 110.205, -106.62, -89.137, 54.679] deg; flange x=154.353 y=-431.082 z=317.99 mm, rx=1.296 ry=2.8485 rz=0.0145 rad
  MoveL speed 250 mm/s, acceleration 1200 mm/s^2 (useActiveTCP=true) feature=Base
    Waypoint L2_H: TCP in base x=120.951 y=-463.337 z=47.814 mm, rx=1.296 ry=2.8485 rz=0.0145 rad; joints [90.81, -90.543, 107.34, -106.612, -89.15, 49.739] deg; flange x=116.95 y=-464.264 z=318.193 mm, rx=1.296 ry=2.8485 rz=0.0145 rad
  MoveL speed 250 mm/s, acceleration 1200 mm/s^2 (useActiveTCP=true) feature=Base
    Waypoint L3_H: TCP in base x=154.133 y=-500.739 z=47.86 mm, rx=1.296 ry=2.8485 rz=0.0145 rad; joints [94.491, -84.421, 100.92, -106.37, -89.139, 53.42] deg; flange x=150.132 y=-501.666 z=318.239 mm, rx=1.296 ry=2.8485 rz=0.0145 rad
  MoveL speed 250 mm/s, acceleration 1200 mm/s^2 (useActiveTCP=true) feature=Base
    Waypoint L4_H: TCP in base x=116.731 y=-533.921 z=48.063 mm, rx=1.296 ry=2.8485 rz=0.0145 rad; joints [90.253, -81.345, 97.368, -105.83, -89.151, 49.181] deg; flange x=112.73 y=-534.848 z=318.442 mm, rx=1.296 ry=2.8485 rz=0.0145 rad
  MoveL speed 250 mm/s, acceleration 1200 mm/s^2 (useActiveTCP=true) feature=Base
    Waypoint L5_H: TCP in base x=83.549 y=-496.518 z=48.017 mm, rx=1.296 ry=2.8485 rz=0.0145 rad; joints [86.432, -87.104, 103.773, -106.421, -89.166, 45.36] deg; flange x=79.548 y=-497.445 z=318.396 mm, rx=1.296 ry=2.8485 rz=0.0145 rad
  MoveL speed 250 mm/s, acceleration 1200 mm/s^2 (useActiveTCP=true) feature=Base
    Waypoint L6_H: TCP in base x=46.146 y=-529.7 z=48.22 mm, rx=1.296 ry=2.8485 rz=0.0145 rad; joints [82.58, -83.248, 99.507, -105.954, -89.185, 41.507] deg; flange x=42.145 y=-530.627 z=318.599 mm, rx=1.296 ry=2.8485 rz=0.0145 rad
  MoveL speed 250 mm/s, acceleration 1200 mm/s^2 (useActiveTCP=true) feature=Base
    Waypoint L7_H: TCP in base x=145.692 y=-641.908 z=48.359 mm, rx=1.296 ry=2.8485 rz=0.0145 rad; joints [92.777, -66.425, 77.805, -101.226, -89.144, 51.706] deg; flange x=141.691 y=-642.835 z=318.738 mm, rx=1.296 ry=2.8485 rz=0.0145 rad
  MoveL speed 250 mm/s, acceleration 1200 mm/s^2 (useActiveTCP=true) feature=Base
    Waypoint L8: TCP in base x=183.095 y=-608.726 z=48.156 mm, rx=1.296 ry=2.8485 rz=0.0145 rad; joints [96.366, -69.532, 82.247, -102.614, -89.136, 55.295] deg; flange x=179.094 y=-609.653 z=318.535 mm, rx=1.296 ry=2.8485 rz=0.0145 rad
  MoveL speed 250 mm/s, acceleration 1200 mm/s^2 (useActiveTCP=true) feature=Base
    Waypoint L9_H: TCP in base x=149.913 y=-571.324 z=48.11 mm, rx=1.296 ry=2.8485 rz=0.0145 rad; joints [93.532, -75.512, 90.226, -104.57, -89.142, 52.461] deg; flange x=145.912 y=-572.25 z=318.489 mm, rx=1.296 ry=2.8485 rz=0.0145 rad
  MoveL speed 250 mm/s, acceleration 1200 mm/s^2 (useActiveTCP=true) feature=Base
    Waypoint L10_H: TCP in base x=187.315 y=-538.142 z=47.907 mm, rx=1.296 ry=2.8485 rz=0.0145 rad; joints [97.601, -78.323, 93.797, -105.391, -89.134, 56.531] deg; flange x=183.314 y=-539.069 z=318.286 mm, rx=1.296 ry=2.8485 rz=0.0145 rad
  MoveL speed 250 mm/s, acceleration 1200 mm/s^2 (useActiveTCP=true) feature=Base
    Waypoint L11_H: TCP in base x=220.497 y=-575.545 z=47.953 mm, rx=1.296 ry=2.8485 rz=0.0145 rad; joints [100.256, -72.166, 85.887, -103.679, -89.131, 59.185] deg; flange x=216.496 y=-576.472 z=318.332 mm, rx=1.296 ry=2.8485 rz=0.0145 rad
  MoveL speed 250 mm/s, acceleration 1200 mm/s^2 (useActiveTCP=true) feature=Base
    Waypoint L12_H: TCP in base x=257.899 y=-542.363 z=47.75 mm, rx=1.296 ry=2.8485 rz=0.0145 rad; joints [104.44, -74.31, 88.769, -104.48, -89.13, 63.37] deg; flange x=253.899 y=-543.29 z=318.129 mm, rx=1.296 ry=2.8485 rz=0.0145 rad
SubProgram Umple_P4_H (keepSynchronizedWithDisk=false)
  MoveJ speed 60 deg/s, acceleration 80 deg/s^2 (useActiveTCP=true)
    Waypoint INTERM_P4_H: TCP in base x=-167.567 y=-286.499 z=168.811 mm, rx=1.2909 ry=2.8479 rz=-0.0144 rad; joints [39.36, -114.131, 107.649, -83.617, -89.01, -1.87] deg; flange x=-170.167 y=-282.588 z=439.18 mm, rx=1.2909 ry=2.8479 rz=-0.0144 rad
    Wait Sleep waitTime=0.5
  MoveJ speed 60 deg/s, acceleration 80 deg/s^2 (useActiveTCP=true)
    Waypoint DEAS_C4_H: TCP in base x=-634.049 y=166.753 z=111.017 mm, rx=1.0761 ry=2.3886 rz=1.0065 rad; joints [-7.715, -31.545, 17.047, -40.87, -122.454, -38.841] deg; flange x=-782.032 y=40.366 z=298.765 mm, rx=1.0761 ry=2.3886 rz=1.0065 rad
    Wait Sleep waitTime=0.5
  MoveL speed 250 mm/s, acceleration 1200 mm/s^2 (useActiveTCP=true) feature=Base
    Waypoint PREL_C4_H: TCP in base x=-580.967 y=215.041 z=41.371 mm, rx=1.0761 ry=2.3886 rz=1.0065 rad; joints [-11.8, -45.21, 53.1, -65.52, -124.71, -42.93] deg; flange x=-728.95 y=88.654 z=229.118 mm, rx=1.0761 ry=2.3886 rz=1.0065 rad
    Wait Sleep waitTime=0.5
    'G40'
  MoveL speed 250 mm/s, acceleration 1200 mm/s^2 (useActiveTCP=true) feature=Base
    Waypoint DEAS_C4_HH: TCP in base x=-634.049 y=166.753 z=111.017 mm, rx=1.0761 ry=2.3886 rz=1.0065 rad; joints [-7.715, -31.545, 17.047, -40.87, -122.454, -38.841] deg; flange x=-782.032 y=40.366 z=298.765 mm, rx=1.0761 ry=2.3886 rz=1.0065 rad
    Wait Sleep waitTime=0.5
  MoveJ speed 60 deg/s, acceleration 80 deg/s^2 (useActiveTCP=true)
    Waypoint INTERMEDIA: TCP in base x=-167.567 y=-286.499 z=168.811 mm, rx=1.2909 ry=2.8479 rz=-0.0144 rad; joints [39.36, -114.131, 107.649, -83.617, -89.01, -1.87] deg; flange x=-170.167 y=-282.588 z=439.18 mm, rx=1.2909 ry=2.8479 rz=-0.0144 rad
    Wait Sleep waitTime=0.5
  MoveJ speed 60 deg/s, acceleration 80 deg/s^2 (useActiveTCP=true)
    Waypoint DEAS_P4_H_FOAIE: TCP in base x=148.18 y=-606.801 z=148.804 mm, rx=2.9838 ry=0.9733 rz=-0.0057 rad; joints [93.749, -72.614, 71.678, -89.283, -90.157, 147.616] deg; flange x=148.852 y=-605.72 z=419.211 mm, rx=2.9838 ry=0.9733 rz=-0.0057 rad
    Wait Sleep waitTime=0.5
  MoveL speed 250 mm/s, acceleration 1200 mm/s^2 (useActiveTCP=true) feature=Base
    Waypoint LAS_P4_H_FOAIE: TCP in base x=147.775 y=-607.367 z=-18.541 mm, rx=2.9838 ry=0.9733 rz=-0.0057 rad; joints [93.708, -68.278, 90.79, -112.731, -90.157, 147.575] deg; flange x=148.447 y=-606.286 z=251.866 mm, rx=2.9838 ry=0.9733 rz=-0.0057 rad
    Wait Sleep waitTime=0.5
    'G 80'
  MoveL speed 250 mm/s, acceleration 1200 mm/s^2 (useActiveTCP=true) feature=Base
    Waypoint DEAS_P4_H: TCP in base x=148.179 y=-606.801 z=148.804 mm, rx=2.9838 ry=0.9733 rz=-0.0056 rad; joints [93.749, -72.614, 71.678, -89.284, -90.157, 147.616] deg; flange x=148.85 y=-605.719 z=419.211 mm, rx=2.9838 ry=0.9733 rz=-0.0056 rad
    Wait Sleep waitTime=0.5
SubProgram Umple_P5_H (keepSynchronizedWithDisk=false)
  MoveJ speed 60 deg/s, acceleration 80 deg/s^2 (useActiveTCP=true)
    Waypoint INTERM_P5_H: TCP in base x=-167.567 y=-286.499 z=168.811 mm, rx=1.2909 ry=2.8479 rz=-0.0144 rad; joints [39.36, -114.131, 107.649, -83.617, -89.01, -1.87] deg; flange x=-170.167 y=-282.588 z=439.18 mm, rx=1.2909 ry=2.8479 rz=-0.0144 rad
    Wait Sleep waitTime=0.5
  MoveJ speed 60 deg/s, acceleration 80 deg/s^2 (useActiveTCP=true)
    Waypoint DEAS_C5_H: TCP in base x=-634.049 y=166.753 z=111.017 mm, rx=1.0761 ry=2.3886 rz=1.0065 rad; joints [-7.715, -31.545, 17.047, -40.87, -122.454, -38.841] deg; flange x=-782.032 y=40.366 z=298.765 mm, rx=1.0761 ry=2.3886 rz=1.0065 rad
    Wait Sleep waitTime=0.5
  MoveL speed 250 mm/s, acceleration 1200 mm/s^2 (useActiveTCP=true) feature=Base
    Waypoint PREL_C5_H: TCP in base x=-580.967 y=215.041 z=41.371 mm, rx=1.0761 ry=2.3886 rz=1.0065 rad; joints [-11.8, -45.21, 53.1, -65.52, -124.71, -42.93] deg; flange x=-728.95 y=88.654 z=229.118 mm, rx=1.0761 ry=2.3886 rz=1.0065 rad
    Wait Sleep waitTime=0.5
    'G40'
  MoveL speed 250 mm/s, acceleration 1200 mm/s^2 (useActiveTCP=true) feature=Base
    Waypoint DEAS_C5_HH: TCP in base x=-634.049 y=166.753 z=111.017 mm, rx=1.0761 ry=2.3886 rz=1.0065 rad; joints [-7.715, -31.545, 17.047, -40.87, -122.454, -38.841] deg; flange x=-782.032 y=40.366 z=298.765 mm, rx=1.0761 ry=2.3886 rz=1.0065 rad
    Wait Sleep waitTime=0.5
  MoveJ speed 60 deg/s, acceleration 80 deg/s^2 (useActiveTCP=true)
    Waypoint inter: TCP in base x=-167.567 y=-286.499 z=168.811 mm, rx=1.2909 ry=2.8479 rz=-0.0144 rad; joints [39.36, -114.131, 107.649, -83.617, -89.01, -1.87] deg; flange x=-170.167 y=-282.588 z=439.18 mm, rx=1.2909 ry=2.8479 rz=-0.0144 rad
    Wait Sleep waitTime=0.5
  MoveJ speed 60 deg/s, acceleration 80 deg/s^2 (useActiveTCP=true)
    Waypoint DEAS_P5_H_FOAIE: TCP in base x=114.998 y=-569.398 z=148.758 mm, rx=2.9838 ry=0.9733 rz=-0.0057 rad; joints [90.678, -78.814, 79.543, -90.957, -90.145, 144.545] deg; flange x=115.67 y=-568.317 z=419.165 mm, rx=2.9838 ry=0.9733 rz=-0.0057 rad
    Wait Sleep waitTime=0.5
  MoveL speed 250 mm/s, acceleration 1200 mm/s^2 (useActiveTCP=true) feature=Base
    Waypoint LAS_P5_H_FOAIE: TCP in base x=114.593 y=-569.965 z=-18.588 mm, rx=2.9838 ry=0.9733 rz=-0.0057 rad; joints [90.636, -73.794, 98.433, -114.866, -90.145, 144.503] deg; flange x=115.265 y=-568.884 z=251.819 mm, rx=2.9838 ry=0.9733 rz=-0.0057 rad
    Wait Sleep waitTime=0.5
    'G 80'
  MoveL speed 250 mm/s, acceleration 1200 mm/s^2 (useActiveTCP=true) feature=Base
    Waypoint DEAS_C5_H_FOAIE: TCP in base x=114.997 y=-569.398 z=148.758 mm, rx=2.9838 ry=0.9733 rz=-0.0056 rad; joints [90.677, -78.814, 79.543, -90.957, -90.145, 144.544] deg; flange x=115.668 y=-568.317 z=419.165 mm, rx=2.9838 ry=0.9733 rz=-0.0056 rad
    Wait Sleep waitTime=0.5
SubProgram Umple_P6_H (keepSynchronizedWithDisk=false)
  MoveJ speed 60 deg/s, acceleration 80 deg/s^2 (useActiveTCP=true)
    Waypoint INTERM_C6_H: TCP in base x=-167.567 y=-286.499 z=168.811 mm, rx=1.2909 ry=2.8479 rz=-0.0144 rad; joints [39.36, -114.131, 107.649, -83.617, -89.01, -1.87] deg; flange x=-170.167 y=-282.588 z=439.18 mm, rx=1.2909 ry=2.8479 rz=-0.0144 rad
    Wait Sleep waitTime=0.5
  MoveJ speed 60 deg/s, acceleration 80 deg/s^2 (useActiveTCP=true)
    Waypoint DEAS_C6_H: TCP in base x=-634.049 y=166.753 z=111.017 mm, rx=1.0761 ry=2.3886 rz=1.0065 rad; joints [-7.715, -31.545, 17.047, -40.87, -122.454, -38.841] deg; flange x=-782.032 y=40.366 z=298.765 mm, rx=1.0761 ry=2.3886 rz=1.0065 rad
    Wait Sleep waitTime=0.5
  MoveL speed 250 mm/s, acceleration 1200 mm/s^2 (useActiveTCP=true) feature=Base
    Waypoint PREL_C6_H: TCP in base x=-580.967 y=215.041 z=41.371 mm, rx=1.0761 ry=2.3886 rz=1.0065 rad; joints [-11.8, -45.21, 53.1, -65.52, -124.71, -42.93] deg; flange x=-728.95 y=88.654 z=229.118 mm, rx=1.0761 ry=2.3886 rz=1.0065 rad
    Wait Sleep waitTime=0.5
    'G40'
  MoveL speed 250 mm/s, acceleration 1200 mm/s^2 (useActiveTCP=true) feature=Base
    Waypoint DEAS_C6_HH: TCP in base x=-634.049 y=166.753 z=111.017 mm, rx=1.0761 ry=2.3886 rz=1.0065 rad; joints [-7.715, -31.545, 17.047, -40.87, -122.454, -38.841] deg; flange x=-782.032 y=40.366 z=298.765 mm, rx=1.0761 ry=2.3886 rz=1.0065 rad
    Wait Sleep waitTime=0.5
  MoveJ speed 60 deg/s, acceleration 80 deg/s^2 (useActiveTCP=true)
    Waypoint INTERMEDIARR: TCP in base x=-167.567 y=-286.499 z=168.811 mm, rx=1.2909 ry=2.8479 rz=-0.0144 rad; joints [39.36, -114.131, 107.649, -83.617, -89.01, -1.87] deg; flange x=-170.167 y=-282.588 z=439.18 mm, rx=1.2909 ry=2.8479 rz=-0.0144 rad
    Wait Sleep waitTime=0.5
  MoveJ speed 60 deg/s, acceleration 80 deg/s^2 (useActiveTCP=true)
    Waypoint DEAS_P6_H_FOAIE: TCP in base x=81.816 y=-531.995 z=148.712 mm, rx=2.9838 ry=0.9733 rz=-0.0057 rad; joints [87.131, -84.729, 86.384, -91.892, -90.131, 140.998] deg; flange x=82.488 y=-530.914 z=419.119 mm, rx=2.9838 ry=0.9733 rz=-0.0057 rad
    Wait Sleep waitTime=0.5
  MoveL speed 250 mm/s, acceleration 1200 mm/s^2 (useActiveTCP=true) feature=Base
    Waypoint LAS_P6_H_FOAIE: TCP in base x=81.411 y=-532.562 z=-18.634 mm, rx=2.9838 ry=0.9733 rz=-0.0057 rad; joints [87.09, -79.208, 105.372, -116.4, -90.131, 140.957] deg; flange x=82.083 y=-531.481 z=251.773 mm, rx=2.9838 ry=0.9733 rz=-0.0057 rad
    Wait Sleep waitTime=0.5
    'G 80'
  MoveL speed 250 mm/s, acceleration 1200 mm/s^2 (useActiveTCP=true) feature=Base
    Waypoint DEAS_C6_H_FOAIE: TCP in base x=81.815 y=-531.995 z=148.711 mm, rx=2.9838 ry=0.9733 rz=-0.0056 rad; joints [87.13, -84.729, 86.385, -91.892, -90.13, 140.997] deg; flange x=82.486 y=-530.914 z=419.118 mm, rx=2.9838 ry=0.9733 rz=-0.0056 rad
    Wait Sleep waitTime=0.5
SubProgram Umple_P7_H (keepSynchronizedWithDisk=false)
  MoveJ speed 60 deg/s, acceleration 80 deg/s^2 (useActiveTCP=true)
    Waypoint INTERMED_P7_H: TCP in base x=-167.567 y=-286.499 z=168.811 mm, rx=1.2909 ry=2.8479 rz=-0.0144 rad; joints [39.36, -114.131, 107.649, -83.617, -89.01, -1.87] deg; flange x=-170.167 y=-282.588 z=439.18 mm, rx=1.2909 ry=2.8479 rz=-0.0144 rad
    Wait Sleep waitTime=0.5
  MoveJ speed 60 deg/s, acceleration 80 deg/s^2 (useActiveTCP=true)
    Waypoint DEAS_C7_H: TCP in base x=-634.049 y=166.753 z=111.017 mm, rx=1.0761 ry=2.3886 rz=1.0065 rad; joints [-7.715, -31.545, 17.047, -40.87, -122.454, -38.841] deg; flange x=-782.032 y=40.366 z=298.765 mm, rx=1.0761 ry=2.3886 rz=1.0065 rad
    Wait Sleep waitTime=0.5
  MoveL speed 250 mm/s, acceleration 1200 mm/s^2 (useActiveTCP=true) feature=Base
    Waypoint PREL_C7_H: TCP in base x=-580.967 y=215.041 z=41.371 mm, rx=1.0761 ry=2.3886 rz=1.0065 rad; joints [-11.8, -45.21, 53.1, -65.52, -124.71, -42.93] deg; flange x=-728.95 y=88.654 z=229.118 mm, rx=1.0761 ry=2.3886 rz=1.0065 rad
    Wait Sleep waitTime=0.5
    'G40'
  MoveL speed 250 mm/s, acceleration 1200 mm/s^2 (useActiveTCP=true) feature=Base
    Waypoint DEAS_C7_HH: TCP in base x=-634.049 y=166.753 z=111.017 mm, rx=1.0761 ry=2.3886 rz=1.0065 rad; joints [-7.715, -31.545, 17.047, -40.87, -122.454, -38.841] deg; flange x=-782.032 y=40.366 z=298.765 mm, rx=1.0761 ry=2.3886 rz=1.0065 rad
    Wait Sleep waitTime=0.5
  MoveJ speed 60 deg/s, acceleration 80 deg/s^2 (useActiveTCP=true)
    Waypoint intermed: TCP in base x=-167.567 y=-286.499 z=168.811 mm, rx=1.2909 ry=2.8479 rz=-0.0144 rad; joints [39.36, -114.131, 107.649, -83.617, -89.01, -1.87] deg; flange x=-170.167 y=-282.588 z=439.18 mm, rx=1.2909 ry=2.8479 rz=-0.0144 rad
    Wait Sleep waitTime=0.5
  MoveJ speed 60 deg/s, acceleration 80 deg/s^2 (useActiveTCP=true)
    Waypoint DEAS_P7_H_FOAIE: TCP in base x=152.4 y=-536.217 z=148.555 mm, rx=1.2912 ry=2.8474 rz=-0.0143 rad; joints [94.246, -82.712, 84.313, -92.475, -89.492, 53.037] deg; flange x=149.701 y=-532.282 z=418.923 mm, rx=1.2912 ry=2.8474 rz=-0.0143 rad
    Wait Sleep waitTime=0.5
  MoveJ speed 60 deg/s, acceleration 80 deg/s^2 (useActiveTCP=true)
    Waypoint LAS_P7_H_FOAIE: TCP in base x=151.995 y=-536.783 z=-18.791 mm, rx=1.2912 ry=2.8474 rz=-0.0143 rad; joints [94.199, -77.279, 103.174, -116.768, -89.491, 52.99] deg; flange x=149.296 y=-532.849 z=251.577 mm, rx=1.2912 ry=2.8474 rz=-0.0143 rad
    Wait Sleep waitTime=0.5
    'G 80'
  MoveL speed 250 mm/s, acceleration 1200 mm/s^2 (useActiveTCP=true) feature=Base
    Waypoint DEAS_C7_H_FOAIE: TCP in base x=152.4 y=-536.217 z=148.555 mm, rx=1.2912 ry=2.8474 rz=-0.0143 rad; joints [94.246, -82.712, 84.313, -92.475, -89.492, 53.037] deg; flange x=149.701 y=-532.282 z=418.923 mm, rx=1.2912 ry=2.8474 rz=-0.0143 rad
SubProgram Desen_T (keepSynchronizedWithDisk=false)
  MoveL speed 250 mm/s, acceleration 1200 mm/s^2 (useActiveTCP=true) feature=Base
    Waypoint l1_T: TCP in base x=224.718 y=-504.961 z=47.704 mm, rx=1.296 ry=2.8485 rz=0.0145 rad; joints [102.033, -80.643, 96.641, -105.983, -89.13, 60.963] deg; flange x=220.717 y=-505.887 z=318.083 mm, rx=1.296 ry=2.8485 rz=0.0145 rad
  MoveL speed 250 mm/s, acceleration 1200 mm/s^2 (useActiveTCP=true) feature=Base
    Waypoint l2_T: TCP in base x=187.315 y=-538.142 z=47.907 mm, rx=1.296 ry=2.8485 rz=0.0145 rad; joints [97.601, -78.323, 93.797, -105.391, -89.134, 56.531] deg; flange x=183.314 y=-539.069 z=318.286 mm, rx=1.296 ry=2.8485 rz=0.0145 rad
  MoveL speed 250 mm/s, acceleration 1200 mm/s^2 (useActiveTCP=true) feature=Base
    Waypoint l3_T: TCP in base x=87.769 y=-425.934 z=47.768 mm, rx=1.296 ry=2.8485 rz=0.0145 rad; joints [86.408, -96.745, 113.088, -106.093, -89.166, 45.336] deg; flange x=83.768 y=-426.861 z=318.147 mm, rx=1.296 ry=2.8485 rz=0.0145 rad
  MoveL speed 250 mm/s, acceleration 1200 mm/s^2 (useActiveTCP=true) feature=Base
    Waypoint l4_T: TCP in base x=50.367 y=-459.116 z=47.971 mm, rx=1.296 ry=2.8485 rz=0.0145 rad; joints [81.952, -92.826, 109.491, -106.351, -89.188, 40.88] deg; flange x=46.366 y=-460.043 z=318.35 mm, rx=1.296 ry=2.8485 rz=0.0145 rad
  MoveL speed 250 mm/s, acceleration 1200 mm/s^2 (useActiveTCP=true) feature=Base
    Waypoint l5_T: TCP in base x=149.913 y=-571.324 z=48.11 mm, rx=1.296 ry=2.8485 rz=0.0145 rad; joints [93.532, -75.512, 90.226, -104.57, -89.142, 52.461] deg; flange x=145.912 y=-572.251 z=318.489 mm, rx=1.296 ry=2.8485 rz=0.0145 rad
  MoveL speed 250 mm/s, acceleration 1200 mm/s^2 (useActiveTCP=true) feature=Base
    Waypoint l6_T: TCP in base x=112.51 y=-604.505 z=48.313 mm, rx=1.296 ry=2.8485 rz=0.0145 rad; joints [89.824, -72.249, 85.906, -103.458, -89.153, 48.753] deg; flange x=108.509 y=-605.432 z=318.692 mm, rx=1.296 ry=2.8485 rz=0.0145 rad
  MoveL speed 250 mm/s, acceleration 1200 mm/s^2 (useActiveTCP=true) feature=Base
    Waypoint l7_T: TCP in base x=145.692 y=-641.908 z=48.359 mm, rx=1.296 ry=2.8485 rz=0.0145 rad; joints [92.777, -66.425, 77.805, -101.226, -89.144, 51.706] deg; flange x=141.691 y=-642.835 z=318.738 mm, rx=1.296 ry=2.8485 rz=0.0145 rad
  MoveL speed 250 mm/s, acceleration 1200 mm/s^2 (useActiveTCP=true) feature=Base
    Waypoint l8_T: TCP in base x=257.9 y=-542.363 z=47.751 mm, rx=1.296 ry=2.8485 rz=0.0145 rad; joints [104.44, -74.31, 88.769, -104.48, -89.13, 63.37] deg; flange x=253.899 y=-543.29 z=318.129 mm, rx=1.296 ry=2.8485 rz=0.0145 rad
SubProgram Umple_P2_T (keepSynchronizedWithDisk=false)
  MoveJ speed 60 deg/s, acceleration 80 deg/s^2 (useActiveTCP=true)
    Waypoint INTERM_P2_T: TCP in base x=-167.567 y=-286.499 z=168.811 mm, rx=1.2909 ry=2.8479 rz=-0.0144 rad; joints [39.36, -114.131, 107.649, -83.617, -89.01, -1.87] deg; flange x=-170.167 y=-282.588 z=439.18 mm, rx=1.2909 ry=2.8479 rz=-0.0144 rad
    Wait Sleep waitTime=0.5
  MoveJ speed 60 deg/s, acceleration 80 deg/s^2 (useActiveTCP=true)
    Waypoint DEAS_P2_T: TCP in base x=-634.049 y=166.753 z=111.017 mm, rx=1.0761 ry=2.3886 rz=1.0065 rad; joints [-7.715, -31.545, 17.047, -40.87, -122.454, -38.841] deg; flange x=-782.032 y=40.366 z=298.765 mm, rx=1.0761 ry=2.3886 rz=1.0065 rad
    Wait Sleep waitTime=0.5
  MoveL speed 250 mm/s, acceleration 1200 mm/s^2 (useActiveTCP=true) feature=Base
    Waypoint PREL_C2_T: TCP in base x=-580.967 y=215.041 z=41.371 mm, rx=1.0761 ry=2.3886 rz=1.0065 rad; joints [-11.8, -45.21, 53.1, -65.52, -124.71, -42.93] deg; flange x=-728.95 y=88.654 z=229.118 mm, rx=1.0761 ry=2.3886 rz=1.0065 rad
    Wait Sleep waitTime=0.5
    'G40'
  MoveL speed 250 mm/s, acceleration 1200 mm/s^2 (useActiveTCP=true) feature=Base
    Waypoint DEAS_C2_T: TCP in base x=-634.049 y=166.753 z=111.017 mm, rx=1.0761 ry=2.3886 rz=1.0065 rad; joints [-7.715, -31.545, 17.047, -40.87, -122.454, -38.841] deg; flange x=-782.032 y=40.366 z=298.765 mm, rx=1.0761 ry=2.3886 rz=1.0065 rad
    Wait Sleep waitTime=0.5
  MoveJ speed 60 deg/s, acceleration 80 deg/s^2 (useActiveTCP=true)
    Waypoint INTERMED: TCP in base x=-167.567 y=-286.499 z=168.811 mm, rx=1.2909 ry=2.8479 rz=-0.0144 rad; joints [39.36, -114.131, 107.649, -83.617, -89.01, -1.87] deg; flange x=-170.167 y=-282.588 z=439.18 mm, rx=1.2909 ry=2.8479 rz=-0.0144 rad
    Wait Sleep waitTime=0.5
  MoveJ speed 60 deg/s, acceleration 80 deg/s^2 (useActiveTCP=true)
    Waypoint DEAS_P2_T_FOAIE: TCP in base x=185.582 y=-573.619 z=148.601 mm, rx=1.2912 ry=2.8474 rz=-0.0143 rad; joints [97.222, -76.393, 76.753, -91.258, -89.538, 56.012] deg; flange x=182.883 y=-569.684 z=418.969 mm, rx=1.2912 ry=2.8474 rz=-0.0143 rad
    Wait Sleep waitTime=0.5
  MoveL speed 250 mm/s, acceleration 1200 mm/s^2 (useActiveTCP=true) feature=Base
    Waypoint LAS_P2_T_FOAIE: TCP in base x=185.177 y=-574.186 z=-18.744 mm, rx=1.2912 ry=2.8474 rz=-0.0143 rad; joints [97.176, -71.555, 95.612, -114.956, -89.537, 55.966] deg; flange x=182.478 y=-570.251 z=251.624 mm, rx=1.2912 ry=2.8474 rz=-0.0143 rad
    Wait Sleep waitTime=0.5
    'G 80'
  MoveL speed 250 mm/s, acceleration 1200 mm/s^2 (useActiveTCP=true) feature=Base
    Waypoint DEAS_P2_T_F: TCP in base x=185.582 y=-573.619 z=148.601 mm, rx=1.2912 ry=2.8474 rz=-0.0143 rad; joints [97.222, -76.393, 76.753, -91.258, -89.538, 56.012] deg; flange x=182.883 y=-569.684 z=418.969 mm, rx=1.2912 ry=2.8474 rz=-0.0143 rad
    Wait Sleep waitTime=0.5
SubProgram Umple_p3_T (keepSynchronizedWithDisk=false)
  MoveJ speed 60 deg/s, acceleration 80 deg/s^2 (useActiveTCP=true)
    Waypoint INTERM_P3_T: TCP in base x=-167.567 y=-286.499 z=168.811 mm, rx=1.2909 ry=2.8479 rz=-0.0144 rad; joints [39.36, -114.131, 107.649, -83.617, -89.01, -1.87] deg; flange x=-170.167 y=-282.588 z=439.18 mm, rx=1.2909 ry=2.8479 rz=-0.0144 rad
    Wait Sleep waitTime=0.5
  MoveJ speed 60 deg/s, acceleration 80 deg/s^2 (useActiveTCP=true)
    Waypoint DEAS_C3_T: TCP in base x=-634.049 y=166.753 z=111.017 mm, rx=1.0761 ry=2.3886 rz=1.0065 rad; joints [-7.715, -31.545, 17.047, -40.87, -122.454, -38.841] deg; flange x=-782.032 y=40.366 z=298.765 mm, rx=1.0761 ry=2.3886 rz=1.0065 rad
    Wait Sleep waitTime=0.5
  MoveL speed 250 mm/s, acceleration 1200 mm/s^2 (useActiveTCP=true) feature=Base
    Waypoint PREL_C3_T: TCP in base x=-580.967 y=215.041 z=41.371 mm, rx=1.0761 ry=2.3886 rz=1.0065 rad; joints [-11.8, -45.21, 53.1, -65.52, -124.71, -42.93] deg; flange x=-728.95 y=88.654 z=229.118 mm, rx=1.0761 ry=2.3886 rz=1.0065 rad
    Wait Sleep waitTime=0.5
    'G40'
  MoveL speed 250 mm/s, acceleration 1200 mm/s^2 (useActiveTCP=true) feature=Base
    Waypoint DEAS_C3_TT: TCP in base x=-634.049 y=166.753 z=111.017 mm, rx=1.0761 ry=2.3886 rz=1.0065 rad; joints [-7.715, -31.545, 17.047, -40.87, -122.454, -38.841] deg; flange x=-782.032 y=40.366 z=298.765 mm, rx=1.0761 ry=2.3886 rz=1.0065 rad
    Wait Sleep waitTime=0.5
  MoveJ speed 60 deg/s, acceleration 80 deg/s^2 (useActiveTCP=true)
    Waypoint INTERMEDD: TCP in base x=-167.567 y=-286.499 z=168.811 mm, rx=1.2909 ry=2.8479 rz=-0.0144 rad; joints [39.36, -114.131, 107.649, -83.617, -89.01, -1.87] deg; flange x=-170.167 y=-282.588 z=439.18 mm, rx=1.2909 ry=2.8479 rz=-0.0144 rad
    Wait Sleep waitTime=0.5
  MoveJ speed 60 deg/s, acceleration 80 deg/s^2 (useActiveTCP=true)
    Waypoint DEAS_P3_T_FOAIE: TCP in base x=148.18 y=-606.801 z=148.804 mm, rx=1.2912 ry=2.8474 rz=-0.0143 rad; joints [93.36, -73.284, 72.725, -90.306, -89.478, 52.15] deg; flange x=145.481 y=-602.866 z=419.172 mm, rx=1.2912 ry=2.8474 rz=-0.0143 rad
    Wait Sleep waitTime=0.5
  MoveL speed 250 mm/s, acceleration 1200 mm/s^2 (useActiveTCP=true) feature=Base
    Waypoint LAS_P3_T_FOAIE: TCP in base x=147.775 y=-607.367 z=-18.542 mm, rx=1.2912 ry=2.8474 rz=-0.0143 rad; joints [93.319, -68.807, 91.722, -113.781, -89.477, 52.109] deg; flange x=145.076 y=-603.433 z=251.826 mm, rx=1.2912 ry=2.8474 rz=-0.0143 rad
    Wait Sleep waitTime=0.5
    'G 80'
  MoveL speed 250 mm/s, acceleration 1200 mm/s^2 (useActiveTCP=true) feature=Base
    Waypoint DEAS_P3_T: TCP in base x=148.18 y=-606.801 z=148.804 mm, rx=1.2912 ry=2.8474 rz=-0.0143 rad; joints [93.36, -73.284, 72.725, -90.306, -89.478, 52.15] deg; flange x=145.481 y=-602.866 z=419.172 mm, rx=1.2912 ry=2.8474 rz=-0.0143 rad
    Wait Sleep waitTime=0.5
SubProgram Umplu_p4_t (keepSynchronizedWithDisk=false)
  MoveJ speed 60 deg/s, acceleration 80 deg/s^2 (useActiveTCP=true)
    Waypoint interm_p4_t: TCP in base x=-167.567 y=-286.499 z=168.811 mm, rx=1.2909 ry=2.8479 rz=-0.0144 rad; joints [39.36, -114.131, 107.649, -83.617, -89.01, -1.87] deg; flange x=-170.167 y=-282.588 z=439.18 mm, rx=1.2909 ry=2.8479 rz=-0.0144 rad
    Wait Sleep waitTime=0.5
  MoveJ speed 60 deg/s, acceleration 80 deg/s^2 (useActiveTCP=true)
    Waypoint deas_c4_T: TCP in base x=-634.049 y=166.753 z=111.017 mm, rx=1.0761 ry=2.3886 rz=1.0065 rad; joints [-7.715, -31.545, 17.047, -40.87, -122.454, -38.841] deg; flange x=-782.032 y=40.366 z=298.765 mm, rx=1.0761 ry=2.3886 rz=1.0065 rad
    Wait Sleep waitTime=0.5
  MoveL speed 250 mm/s, acceleration 1200 mm/s^2 (useActiveTCP=true) feature=Base
    Waypoint PREL_C4_T: TCP in base x=-580.967 y=215.041 z=41.371 mm, rx=1.0761 ry=2.3886 rz=1.0065 rad; joints [-11.8, -45.21, 53.1, -65.52, -124.71, -42.93] deg; flange x=-728.95 y=88.654 z=229.118 mm, rx=1.0761 ry=2.3886 rz=1.0065 rad
    Wait Sleep waitTime=0.5
    'G40'
  MoveL speed 250 mm/s, acceleration 1200 mm/s^2 (useActiveTCP=true) feature=Base
    Waypoint DEAS_C4_T: TCP in base x=-634.049 y=166.753 z=111.017 mm, rx=1.0761 ry=2.3886 rz=1.0065 rad; joints [-7.715, -31.545, 17.047, -40.87, -122.454, -38.841] deg; flange x=-782.032 y=40.366 z=298.765 mm, rx=1.0761 ry=2.3886 rz=1.0065 rad
    Wait Sleep waitTime=0.5
  MoveJ speed 60 deg/s, acceleration 80 deg/s^2 (useActiveTCP=true)
    Waypoint INTERMEDIAR: TCP in base x=-167.567 y=-286.499 z=168.811 mm, rx=1.2909 ry=2.8479 rz=-0.0144 rad; joints [39.36, -114.131, 107.649, -83.617, -89.01, -1.87] deg; flange x=-170.167 y=-282.588 z=439.18 mm, rx=1.2909 ry=2.8479 rz=-0.0144 rad
    Wait Sleep waitTime=0.5
  MoveJ speed 60 deg/s, acceleration 80 deg/s^2 (useActiveTCP=true)
    Waypoint DEAS_P4_T_FOAIE: TCP in base x=152.4 y=-536.216 z=148.555 mm, rx=2.9838 ry=0.9733 rz=-0.0057 rad; joints [94.678, -82.056, 83.397, -91.557, -90.161, 148.545] deg; flange x=153.072 y=-535.136 z=418.962 mm, rx=2.9838 ry=0.9733 rz=-0.0057 rad
    Wait Sleep waitTime=0.5
  MoveL speed 250 mm/s, acceleration 1200 mm/s^2 (useActiveTCP=true) feature=Base
    Waypoint LAS_P4_T_FOAIE: TCP in base x=151.995 y=-536.783 z=-18.791 mm, rx=2.9838 ry=0.9733 rz=-0.0057 rad; joints [94.631, -76.741, 102.307, -115.782, -90.16, 148.498] deg; flange x=152.667 y=-535.702 z=251.616 mm, rx=2.9838 ry=0.9733 rz=-0.0057 rad
    Wait Sleep waitTime=0.5
    'G 80'
  MoveL speed 250 mm/s, acceleration 1200 mm/s^2 (useActiveTCP=true) feature=Base
    Waypoint DEAS_P4_T: TCP in base x=152.4 y=-536.216 z=148.555 mm, rx=2.9838 ry=0.9733 rz=-0.0057 rad; joints [94.678, -82.056, 83.397, -91.557, -90.161, 148.545] deg; flange x=153.072 y=-535.136 z=418.962 mm, rx=2.9838 ry=0.9733 rz=-0.0057 rad
    Wait Sleep waitTime=0.5
SubProgram Umplu_p5_T (keepSynchronizedWithDisk=false)
  MoveJ speed 60 deg/s, acceleration 80 deg/s^2 (useActiveTCP=true)
    Waypoint INTERM_P5_T: TCP in base x=-167.567 y=-286.499 z=168.811 mm, rx=1.2909 ry=2.8479 rz=-0.0144 rad; joints [39.36, -114.131, 107.649, -83.617, -89.01, -1.87] deg; flange x=-170.167 y=-282.588 z=439.18 mm, rx=1.2909 ry=2.8479 rz=-0.0144 rad
    Wait Sleep waitTime=0.5
  MoveJ speed 60 deg/s, acceleration 80 deg/s^2 (useActiveTCP=true)
    Waypoint DEAS_C5_T: TCP in base x=-634.049 y=166.753 z=111.017 mm, rx=1.0761 ry=2.3886 rz=1.0065 rad; joints [-7.715, -31.545, 17.047, -40.87, -122.454, -38.841] deg; flange x=-782.032 y=40.366 z=298.765 mm, rx=1.0761 ry=2.3886 rz=1.0065 rad
    Wait Sleep waitTime=0.5
  MoveL speed 250 mm/s, acceleration 1200 mm/s^2 (useActiveTCP=true) feature=Base
    Waypoint PREL_C5_T: TCP in base x=-580.967 y=215.041 z=41.371 mm, rx=1.0761 ry=2.3886 rz=1.0065 rad; joints [-11.8, -45.21, 53.1, -65.52, -124.71, -42.93] deg; flange x=-728.95 y=88.654 z=229.118 mm, rx=1.0761 ry=2.3886 rz=1.0065 rad
    Wait Sleep waitTime=0.5
    'G40'
  MoveL speed 250 mm/s, acceleration 1200 mm/s^2 (useActiveTCP=true) feature=Base
    Waypoint DEAS_C5_TT: TCP in base x=-634.049 y=166.753 z=111.017 mm, rx=1.0761 ry=2.3886 rz=1.0065 rad; joints [-7.715, -31.545, 17.047, -40.87, -122.454, -38.841] deg; flange x=-782.032 y=40.366 z=298.765 mm, rx=1.0761 ry=2.3886 rz=1.0065 rad
    Wait Sleep waitTime=0.5
  MoveJ speed 60 deg/s, acceleration 80 deg/s^2 (useActiveTCP=true)
    Waypoint INter: TCP in base x=-167.567 y=-286.499 z=168.811 mm, rx=1.2909 ry=2.8479 rz=-0.0144 rad; joints [39.36, -114.131, 107.649, -83.617, -89.01, -1.87] deg; flange x=-170.167 y=-282.588 z=439.18 mm, rx=1.2909 ry=2.8479 rz=-0.0144 rad
    Wait Sleep waitTime=0.5
  MoveJ speed 60 deg/s, acceleration 80 deg/s^2 (useActiveTCP=true)
    Waypoint DEAS_P5_T_FOAIE: TCP in base x=119.218 y=-498.814 z=148.508 mm, rx=2.9838 ry=0.9733 rz=-0.0057 rad; joints [91.258, -88.215, 90.13, -92.141, -90.147, 145.124] deg; flange x=119.89 y=-497.733 z=418.915 mm, rx=2.9838 ry=0.9733 rz=-0.0057 rad
    Wait Sleep waitTime=0.5
  MoveL speed 250 mm/s, acceleration 1200 mm/s^2 (useActiveTCP=true) feature=Base
    Waypoint LAS_C5_T_FOAIE: TCP in base x=118.813 y=-499.381 z=-18.837 mm, rx=2.9838 ry=0.9733 rz=-0.0057 rad; joints [91.21, -82.47, 109.293, -117.049, -90.147, 145.077] deg; flange x=119.485 y=-498.3 z=251.57 mm, rx=2.9838 ry=0.9733 rz=-0.0057 rad
    Wait Sleep waitTime=0.5
    'G 80'
  MoveL speed 250 mm/s, acceleration 1200 mm/s^2 (useActiveTCP=true) feature=Base
    Waypoint DEAS_P5: TCP in base x=119.218 y=-498.814 z=148.508 mm, rx=2.9838 ry=0.9733 rz=-0.0057 rad; joints [91.258, -88.215, 90.13, -92.141, -90.147, 145.124] deg; flange x=119.89 y=-497.733 z=418.915 mm, rx=2.9838 ry=0.9733 rz=-0.0057 rad
    Wait Sleep waitTime=0.5
SubProgram Umple_P6_T (keepSynchronizedWithDisk=false)
  MoveJ speed 60 deg/s, acceleration 80 deg/s^2 (useActiveTCP=true)
    Waypoint INTERM_C6_T: TCP in base x=-167.567 y=-286.499 z=168.811 mm, rx=1.2909 ry=2.8479 rz=-0.0144 rad; joints [39.36, -114.131, 107.649, -83.617, -89.01, -1.87] deg; flange x=-170.167 y=-282.588 z=439.18 mm, rx=1.2909 ry=2.8479 rz=-0.0144 rad
    Wait Sleep waitTime=0.5
  MoveJ speed 60 deg/s, acceleration 80 deg/s^2 (useActiveTCP=true)
    Waypoint DEAS_C6_T: TCP in base x=-634.049 y=166.753 z=111.017 mm, rx=1.0761 ry=2.3886 rz=1.0065 rad; joints [-7.715, -31.545, 17.047, -40.87, -122.454, -38.841] deg; flange x=-782.032 y=40.366 z=298.765 mm, rx=1.0761 ry=2.3886 rz=1.0065 rad
    Wait Sleep waitTime=0.5
  MoveL speed 250 mm/s, acceleration 1200 mm/s^2 (useActiveTCP=true) feature=Base
    Waypoint PREL_C6_T: TCP in base x=-580.967 y=215.041 z=41.371 mm, rx=1.0761 ry=2.3886 rz=1.0065 rad; joints [-11.8, -45.21, 53.1, -65.52, -124.71, -42.93] deg; flange x=-728.95 y=88.654 z=229.118 mm, rx=1.0761 ry=2.3886 rz=1.0065 rad
    Wait Sleep waitTime=0.5
    'G40'
  MoveL speed 250 mm/s, acceleration 1200 mm/s^2 (useActiveTCP=true) feature=Base
    Waypoint DEAS_C6_TT: TCP in base x=-634.049 y=166.753 z=111.017 mm, rx=1.0761 ry=2.3886 rz=1.0065 rad; joints [-7.715, -31.545, 17.047, -40.87, -122.454, -38.841] deg; flange x=-782.032 y=40.366 z=298.765 mm, rx=1.0761 ry=2.3886 rz=1.0065 rad
    Wait Sleep waitTime=0.5
  MoveJ speed 60 deg/s, acceleration 80 deg/s^2 (useActiveTCP=true)
    Waypoint INTERME: TCP in base x=-167.567 y=-286.499 z=168.811 mm, rx=1.2909 ry=2.8479 rz=-0.0144 rad; joints [39.36, -114.131, 107.649, -83.617, -89.01, -1.87] deg; flange x=-170.167 y=-282.588 z=439.18 mm, rx=1.2909 ry=2.8479 rz=-0.0144 rad
    Wait Sleep waitTime=0.5
  MoveJ speed 60 deg/s, acceleration 80 deg/s^2 (useActiveTCP=true)
    Waypoint DEAS_P6_T_FOAIE: TCP in base x=86.036 y=-461.411 z=148.462 mm, rx=2.9838 ry=0.9733 rz=-0.0057 rad; joints [87.216, -94.247, 96.031, -92.02, -90.131, 141.083] deg; flange x=86.708 y=-460.33 z=418.869 mm, rx=2.9838 ry=0.9733 rz=-0.0057 rad
    Wait Sleep waitTime=0.5
  MoveL speed 250 mm/s, acceleration 1200 mm/s^2 (useActiveTCP=true) feature=Base
    Waypoint LAS_C6_T_FOAIE: TCP in base x=85.631 y=-461.978 z=-18.883 mm, rx=2.9838 ry=0.9733 rz=-0.0057 rad; joints [87.169, -88.268, 115.671, -117.639, -90.131, 141.036] deg; flange x=86.303 y=-460.897 z=251.524 mm, rx=2.9838 ry=0.9733 rz=-0.0057 rad
    Wait Sleep waitTime=0.5
    'G 80'
  MoveL speed 250 mm/s, acceleration 1200 mm/s^2 (useActiveTCP=true) feature=Base
    Waypoint DEAS_P6_T: TCP in base x=86.036 y=-461.411 z=148.462 mm, rx=2.9838 ry=0.9733 rz=-0.0057 rad; joints [87.216, -94.247, 96.031, -92.02, -90.131, 141.083] deg; flange x=86.708 y=-460.33 z=418.869 mm, rx=2.9838 ry=0.9733 rz=-0.0057 rad
    Wait Sleep waitTime=0.5
